DATA_BLOCK "G177M"
TITLE =DBG177M  COOLING / HEATING GERM 4
//COPYRIGHT:    (C) 2009  BUHLER AG, CH-9240 UZWIL, SWITZERLAND
//
//PRODUCT:      WinCoS_BIW01_09
//
//TITLE:        COOLING / HEATING GERM 4
//                Machine group DB
//                Maschinengruppen-DB
//
//-------------------------------------------------------------------------
//
//IDENT:        AUTHOR:             DEPT:             DATE:
//
//P01_DB277.1.0 K.Renz              CSB41             13.Jan.2010
//              1st Release
//
//-------------------------------------------------------------------------
//
//PURPOSE:
//
//MANUAL :
//
//RESTRICTIONS:
//
//-------------------------------------------------------------------------
AUTHOR : KR
FAMILY : USW
NAME : DBG177M
VERSION : 0.0

"G177M_Code"
BEGIN
   Gr.FcCode := 0;
   Gr.Spare2 := 0;
   Gr.Spare4 := 0;
   Gr.Spare6 := 0;
   Gr.OutEmptyingTime := 0;
   Gr.ChangeBit.spare := B#16#0;
   Gr.ChangeBit.CBit1 := FALSE;
   Gr.ChangeBit.CBit2 := FALSE;
   Gr.ChangeBit.CBit3 := FALSE;
   Gr.ChangeBit.CBit4 := FALSE;
   Gr.StCode := 0;
   Gr.InEnableGr := FALSE;
   Gr.CmdContinue := FALSE;
   Gr.CmdRestartIdling := FALSE;
   Gr.InReleaseEmptyingTime := FALSE;
   Gr.InFeeding := FALSE;
   Gr.InOutAutostartMan := FALSE;
   Gr.InPreStart := FALSE;
   Gr.CmdManualOff := FALSE;
   Gr.CmdOff := FALSE;
   Gr.CmdOn := FALSE;
   Gr.CmdNext := FALSE;
   Gr.CmdFaultReset := FALSE;
   Gr.InOccupied := FALSE;
   Gr.InManual := FALSE;
   Gr.InLoadedSec := FALSE;
   Gr.InSeqStop := FALSE;
   Gr.ModePassive := FALSE;
   Gr.ModeActive := FALSE;
   Gr.ModeIdling := FALSE;
   Gr.spare163 := FALSE;
   Gr.spare164 := FALSE;
   Gr.spare165 := FALSE;
   Gr.spare166 := FALSE;
   Gr.spare167 := FALSE;
   Gr.StStopped := FALSE;
   Gr.StStarting := FALSE;
   Gr.StStarted := FALSE;
   Gr.StStopping := FALSE;
   Gr.StFault := FALSE;
   Gr.OutLoaded := FALSE;
   Gr.OutWarning := FALSE;
   Gr.OutFeeding := FALSE;
   Gr.OutEnableEl := FALSE;
   Gr.OutEnable1 := FALSE;
   Gr.OutHWStop := FALSE;
   Gr.OutDPFault := FALSE;
   Gr.OutAutostart := FALSE;
   Gr.OutManual := FALSE;
   Gr.OutHornOn := FALSE;
   Gr.OutEnablePrevGr := FALSE;
   Gr.VarStopped := FALSE;
   Gr.VarStarted := FALSE;
   Gr.VarFault := FALSE;
   Gr.VarStartwarning := FALSE;
   Gr.VarFlag1s := FALSE;
   Gr.OutEmptyingTimeDone := FALSE;
   Gr.OutNewWay := FALSE;
   Gr.OutSeqStop := FALSE;
   Gr.OutIdlingTime := 0;
   Gr.InCodePreselect := 0;
   Gr.InLine := 3;
   Gr.InCode := 0;
   Gr.OutCode := 0;
   Gr.Par.ParObjectNo := 17700;
   Gr.Par.ParMgr := TRUE;
   Gr.Par.ParWgr := FALSE;
   Gr.Par.ParGgr := FALSE;
   Gr.Par.ParHornCode := 5;
   Gr.Par.ParIdling := 2;
   Gr.Par.ParEmptyingTime := 0;
   Gr.Par.Para1_0 := FALSE;
   Gr.Par.Para1_1 := FALSE;
   Gr.Par.Para1_2 := FALSE;
   Gr.Par.Para1_3 := FALSE;
   Gr.Par.Para1_4 := FALSE;
   Gr.Par.Para1_5 := FALSE;
   Gr.Par.Para1_6 := FALSE;
   Gr.Par.Para1_7 := FALSE;
   Gr.Par.Para1_8 := FALSE;
   Gr.Par.Para1_9 := FALSE;
   Gr.Par.Para1_10 := FALSE;
   Gr.Par.Para1_11 := FALSE;
   Gr.Par.Para1_12 := FALSE;
   Gr.Par.Para1_13 := FALSE;
   Gr.Par.Para1_14 := FALSE;
   Gr.Par.Para1_15 := FALSE;
   Gr.Par.Para2 := 0;
   Gr.Par.Para3 := 0;
   Gr.Par.Para4 := 0;
   Gr.Par.Para5 := 0;
   InOutValue1 := L#0;
   InOutValue2 := L#0;
   OutWayConflict := FALSE;
   OutSelectionOk := FALSE;
   CmdNewValue := FALSE;
   CmdNewJob := FALSE;
   OutCodeOK := FALSE;
   InEndOfJob := FALSE;
   staWayOk := FALSE;
   EdgeStartRelease := FALSE;
   USW8 := FALSE;
   USW9 := FALSE;
   USW10 := FALSE;
   USW11 := FALSE;
   USW12 := FALSE;
   USW13 := FALSE;
   USW14 := FALSE;
   USW15 := FALSE;
   A_2445_QXV21.StCode := 0;
   A_2445_QXV21.InEnableRev := FALSE;
   A_2445_QXV21.InEnableFwd := FALSE;
   A_2445_QXV21.InSlow := FALSE;
   A_2445_QXV21.InpRunSlow := FALSE;
   A_2445_QXV21.InpRunFast := FALSE;
   A_2445_QXV21.InpRunRev := FALSE;
   A_2445_QXV21.InpRunFwd := FALSE;
   A_2445_QXV21.InpFaultDev := FALSE;
   A_2445_QXV21.CmdOff := FALSE;
   A_2445_QXV21.CmdOn := FALSE;
   A_2445_QXV21.CmdNext := FALSE;
   A_2445_QXV21.CmdFaultReset := FALSE;
   A_2445_QXV21.InLocal := FALSE;
   A_2445_QXV21.InManual := FALSE;
   A_2445_QXV21.InReport := FALSE;
   A_2445_QXV21.InSeqStop := FALSE;
   A_2445_QXV21.InHWStop := FALSE;
   A_2445_QXV21.InDPFault := FALSE;
   A_2445_QXV21.OutIdling := FALSE;
   A_2445_QXV21.OutpRunSlow := FALSE;
   A_2445_QXV21.OutpRunFast := FALSE;
   A_2445_QXV21.OutpRunRev := FALSE;
   A_2445_QXV21.OutpRunFwd := FALSE;
   A_2445_QXV21.OutpFaultReset := FALSE;
   A_2445_QXV21.StStopped := FALSE;
   A_2445_QXV21.StStarting := FALSE;
   A_2445_QXV21.StStartedFwd := FALSE;
   A_2445_QXV21.StStopping := FALSE;
   A_2445_QXV21.StFault := FALSE;
   A_2445_QXV21.StStartedRev := FALSE;
   A_2445_QXV21.InOutManSlow := FALSE;
   A_2445_QXV21.InOutManRev := FALSE;
   A_2445_QXV21.OutAlarmNrLog := 0;
   A_2445_QXV21.Par.ParObjectNo := 17701;
   A_2445_QXV21.Par.ParMsgType := 7053;
   A_2445_QXV21.Par.ParHornCode := 5;
   A_2445_QXV21.Par.ParLogOff := FALSE;
   A_2445_QXV21.Par.ParManual := TRUE;
   A_2445_QXV21.Par.ParRestartDelay := FALSE;
   A_2445_QXV21.Par.Par2Speed := FALSE;
   A_2445_QXV21.Par.ParHeavyStartup := FALSE;
   A_2445_QXV21.Par.spare45 := FALSE;
   A_2445_QXV21.Par.spare46 := FALSE;
   A_2445_QXV21.Par.OutEdgeFaultReset := FALSE;
   A_2445_QXV21.Par.OutDelayFault := FALSE;
   A_2445_QXV21.Par.OutFlagFaultDev := FALSE;
   A_2445_QXV21.Par.ParMonTime := 20;
   A_2445_QXV21.Par.ParStartingTime := 20;
   A_2445_QXV21.Par.ParStoppingTime := 0;
   A_2445_QXV21.Par.ParIdlingTime := 0;
   A_2445_QXV21.Par.ParDelayTime := 10;
   A_2445_QXV21.Par.OutMonTime := 0;
   A_2445_QXV21.Par.OutTransitionTime := 0;
   A_2445_QXV21.Par.OutDelayTime := 0;
   A_2445_QXV21.Par.InOutManPulseLen := 0;
   A_2445_QXV21AI.StCode := 2;
   A_2445_QXV21AI.InMonLL := FALSE;
   A_2445_QXV21AI.InMonL := FALSE;
   A_2445_QXV21AI.InMonMid := FALSE;
   A_2445_QXV21AI.InMonH := FALSE;
   A_2445_QXV21AI.InMonHH := FALSE;
   A_2445_QXV21AI.spare0205 := FALSE;
   A_2445_QXV21AI.InpFaultAI := FALSE;
   A_2445_QXV21AI.InpFaultDev := FALSE;
   A_2445_QXV21AI.InHWStop := FALSE;
   A_2445_QXV21AI.InDPFault := FALSE;
   A_2445_QXV21AI.InDisable := FALSE;
   A_2445_QXV21AI.CmdFaultReset := FALSE;
   A_2445_QXV21AI.InLocal := FALSE;
   A_2445_QXV21AI.spare0305 := FALSE;
   A_2445_QXV21AI.InReport := FALSE;
   A_2445_QXV21AI.spare0307 := FALSE;
   A_2445_QXV21AI.OutLL := FALSE;
   A_2445_QXV21AI.OutL := FALSE;
   A_2445_QXV21AI.OutH := FALSE;
   A_2445_QXV21AI.OutHH := FALSE;
   A_2445_QXV21AI.OutOverflow := FALSE;
   A_2445_QXV21AI.spare0405 := FALSE;
   A_2445_QXV21AI.OutFaultAI := FALSE;
   A_2445_QXV21AI.spare0407 := FALSE;
   A_2445_QXV21AI.StLL := FALSE;
   A_2445_QXV21AI.StL := FALSE;
   A_2445_QXV21AI.StMid := FALSE;
   A_2445_QXV21AI.StH := FALSE;
   A_2445_QXV21AI.StHH := FALSE;
   A_2445_QXV21AI.StFaultAI := FALSE;
   A_2445_QXV21AI.OutWarning := FALSE;
   A_2445_QXV21AI.OutFaulted := FALSE;
   A_2445_QXV21AI.InpValue := 0;
   A_2445_QXV21AI.OutValuePc := 0;
   A_2445_QXV21AI.OutValueUnits := L#0;
   A_2445_QXV21AI.Msg.WarningDoneLL := FALSE;
   A_2445_QXV21AI.Msg.WarningDoneL := FALSE;
   A_2445_QXV21AI.Msg.WarningDoneMid := FALSE;
   A_2445_QXV21AI.Msg.WarningDoneH := FALSE;
   A_2445_QXV21AI.Msg.WarningDoneHH := FALSE;
   A_2445_QXV21AI.Msg.FaultDoneLL := FALSE;
   A_2445_QXV21AI.Msg.FaultDoneL := FALSE;
   A_2445_QXV21AI.Msg.FaultDoneMid := FALSE;
   A_2445_QXV21AI.Msg.FaultDoneH := FALSE;
   A_2445_QXV21AI.Msg.FaultDoneHH := FALSE;
   A_2445_QXV21AI.Msg.FaultDoneDev := FALSE;
   A_2445_QXV21AI.Msg.FaultDoneAI := FALSE;
   A_2445_QXV21AI.OutAlarmNrLog := 0;
   A_2445_QXV21AI.Par.ParObjectNo := 17702;
   A_2445_QXV21AI.Par.ParMsgType := 7252;
   A_2445_QXV21AI.Par.ParHornCode := 0;
   A_2445_QXV21AI.Par.ParLogOff := FALSE;
   A_2445_QXV21AI.Par.ParSpare0401 := FALSE;
   A_2445_QXV21AI.Par.ParValueByUser := FALSE;
   A_2445_QXV21AI.Par.ParLimitsPc := TRUE;
   A_2445_QXV21AI.Par.ParWago := FALSE;
   A_2445_QXV21AI.Par.ParNoHornByWarning := FALSE;
   A_2445_QXV21AI.Par.ParWarningLL := FALSE;
   A_2445_QXV21AI.Par.ParWarningL := FALSE;
   A_2445_QXV21AI.Par.ParWarningMid := FALSE;
   A_2445_QXV21AI.Par.ParWarningH := FALSE;
   A_2445_QXV21AI.Par.ParWarningHH := FALSE;
   A_2445_QXV21AI.Par.ParPreAlarmLL := FALSE;
   A_2445_QXV21AI.Par.ParPreAlarmL := FALSE;
   A_2445_QXV21AI.Par.ParPreAlarmMid := FALSE;
   A_2445_QXV21AI.Par.ParPreAlarmH := FALSE;
   A_2445_QXV21AI.Par.ParPreAlarmHH := FALSE;
   A_2445_QXV21AI.Par.ParUnitsByZeroDigit := L#0;
   A_2445_QXV21AI.Par.ParUnitsByMaxDigit := L#10000;
   A_2445_QXV21AI.Par.ParUnitsBy100Pc := L#10000;
   A_2445_QXV21AI.Par.ParLimitLL := L#0;
   A_2445_QXV21AI.Par.ParLimitL := L#2000;
   A_2445_QXV21AI.Par.ParLimitH := L#8000;
   A_2445_QXV21AI.Par.ParLimitHH := L#10000;
   A_2445_QXV21AI.Par.ParMonTimeLL := 0;
   A_2445_QXV21AI.Par.ParMonTimeL := 50;
   A_2445_QXV21AI.Par.ParMonTimeMid := 0;
   A_2445_QXV21AI.Par.ParMonTimeH := 30;
   A_2445_QXV21AI.Par.ParMonTimeHH := 0;
   A_2445_QXV21AI.Par.ParDelayTimeDown := 10;
   A_2445_QXV21AI.Par.ParDelayTimeUp := 10;
   A_2445_QXV21AI.Par.ParDelayTime := 0;
   A_2445_QXV21AI.Par.OutMonTimeLL := 0;
   A_2445_QXV21AI.Par.OutMonTimeL := 50;
   A_2445_QXV21AI.Par.OutMonTimeMid := 0;
   A_2445_QXV21AI.Par.OutMonTimeH := 0;
   A_2445_QXV21AI.Par.OutMonTimeHH := 0;
   A_2445_QXV21AI.Par.OutDelayTimeDown := 0;
   A_2445_QXV21AI.Par.OutDelayTimeUp := 0;
   A_2445_QXV21AI.Par.OutDelayTime := 0;
   A_2445_QXV21AI.Par.Spare66 := 0;
   A_2445_QXV21AO.StCode := 0;
   A_2445_QXV21AO.InDisable := FALSE;
   A_2445_QXV21AO.spare0201 := FALSE;
   A_2445_QXV21AO.spare0202 := FALSE;
   A_2445_QXV21AO.spare0203 := FALSE;
   A_2445_QXV21AO.spare0204 := FALSE;
   A_2445_QXV21AO.spare0205 := FALSE;
   A_2445_QXV21AO.spare0206 := FALSE;
   A_2445_QXV21AO.InpFaultDev := FALSE;
   A_2445_QXV21AO.spare0300 := FALSE;
   A_2445_QXV21AO.spare0301 := FALSE;
   A_2445_QXV21AO.spare0302 := FALSE;
   A_2445_QXV21AO.CmdFaultReset := FALSE;
   A_2445_QXV21AO.InLocal := FALSE;
   A_2445_QXV21AO.InManual := FALSE;
   A_2445_QXV21AO.InReport := FALSE;
   A_2445_QXV21AO.spare0307 := FALSE;
   A_2445_QXV21AO.InHWStop := FALSE;
   A_2445_QXV21AO.InDPFault := FALSE;
   A_2445_QXV21AO.spare0402 := FALSE;
   A_2445_QXV21AO.spare0403 := FALSE;
   A_2445_QXV21AO.spare0404 := FALSE;
   A_2445_QXV21AO.OutpFaultReset := FALSE;
   A_2445_QXV21AO.OutMin := FALSE;
   A_2445_QXV21AO.OutMax := FALSE;
   A_2445_QXV21AO.StOff := FALSE;
   A_2445_QXV21AO.spare0501 := FALSE;
   A_2445_QXV21AO.StOn := FALSE;
   A_2445_QXV21AO.spare0503 := FALSE;
   A_2445_QXV21AO.StFault := FALSE;
   A_2445_QXV21AO.OutpValue := 0;
   A_2445_QXV21AO.InOutValuePc := 0;
   A_2445_QXV21AO.InOutValueUnits := L#0;
   A_2445_QXV21AO.ASW := L#0;
   A_2445_QXV21AO.OutAlarmNrLog := 0;
   A_2445_QXV21AO.Par.ParObjectNo := 17703;
   A_2445_QXV21AO.Par.ParMsgType := 7241;
   A_2445_QXV21AO.Par.ParHornCode := 5;
   A_2445_QXV21AO.Par.ParLogOff := FALSE;
   A_2445_QXV21AO.Par.ParFU := FALSE;
   A_2445_QXV21AO.Par.ParValuePc := TRUE;
   A_2445_QXV21AO.Par.ParLimitsPc := TRUE;
   A_2445_QXV21AO.Par.ParWago := FALSE;
   A_2445_QXV21AO.Par.ParUnitsByZeroDigit := L#0;
   A_2445_QXV21AO.Par.ParUnitsByMaxDigit := L#27648;
   A_2445_QXV21AO.Par.ParUnitsBy100Pc := L#10000;
   A_2445_QXV21AO.Par.ParLimitMin := L#0;
   A_2445_QXV21AO.Par.ParLimitMax := L#27648;
   A_2445_QXV21AO.Par.ParDelayTime := 30;
   A_2445_QXV21AO.Par.OutDelayTime := 0;
   A_2445_QXV21I1.StCode := 0;
   A_2445_QXV21I1.InMonTrue := FALSE;
   A_2445_QXV21I1.InMonFalse := FALSE;
   A_2445_QXV21I1.InPreAlarmTrue := FALSE;
   A_2445_QXV21I1.InPreAlarmFalse := FALSE;
   A_2445_QXV21I1.InStopTrueTime := FALSE;
   A_2445_QXV21I1.InStopFalseTime := FALSE;
   A_2445_QXV21I1.InpTrue := FALSE;
   A_2445_QXV21I1.InpFaultDev := FALSE;
   A_2445_QXV21I1.CmdRstTrueTime := FALSE;
   A_2445_QXV21I1.CmdRstFalseTime := FALSE;
   A_2445_QXV21I1.CmdRunTimeoutTime := FALSE;
   A_2445_QXV21I1.CmdFaultReset := FALSE;
   A_2445_QXV21I1.InLocal := FALSE;
   A_2445_QXV21I1.spare0305 := FALSE;
   A_2445_QXV21I1.InReport := FALSE;
   A_2445_QXV21I1.OutTimeoutTime := FALSE;
   A_2445_QXV21I1.InHWStop := FALSE;
   A_2445_QXV21I1.InDPFault := FALSE;
   A_2445_QXV21I1.OutPreAlarmTrue := FALSE;
   A_2445_QXV21I1.OutPreAlarmFalse := FALSE;
   A_2445_QXV21I1.OutFlagPos := FALSE;
   A_2445_QXV21I1.OutFlagNeg := FALSE;
   A_2445_QXV21I1.OutpFaultReset := FALSE;
   A_2445_QXV21I1.OutTrue := FALSE;
   A_2445_QXV21I1.StFalse := FALSE;
   A_2445_QXV21I1.StCtoTrue := FALSE;
   A_2445_QXV21I1.StTrue := FALSE;
   A_2445_QXV21I1.StCtoFalse := FALSE;
   A_2445_QXV21I1.StFault := FALSE;
   A_2445_QXV21I1.OutAlarmNrLog := 0;
   A_2445_QXV21I1.Par.ParObjectNo := 17704;
   A_2445_QXV21I1.Par.ParMsgType := 7163;
   A_2445_QXV21I1.Par.ParHornCode := 5;
   A_2445_QXV21I1.Par.ParLogOff := FALSE;
   A_2445_QXV21I1.Par.spare0401 := FALSE;
   A_2445_QXV21I1.Par.Par2WorkingCond := FALSE;
   A_2445_QXV21I1.Par.ParFaultRetry := FALSE;
   A_2445_QXV21I1.Par.ParBinLevel := FALSE;
   A_2445_QXV21I1.Par.ParDelayChange := 20;
   A_2445_QXV21I1.Par.ParDelayTrue := 10;
   A_2445_QXV21I1.Par.ParDelayFalse := 0;
   A_2445_QXV21I1.Par.ParTimeoutTrue := 0;
   A_2445_QXV21I1.Par.ParTimeoutFalse := 0;
   A_2445_QXV21I1.Par.OutMonTime := 0;
   A_2445_QXV21I1.Par.OutTransitionTime := 0;
   A_2445_QXV21I1.Par.OutMonTrue := FALSE;
   A_2445_QXV21I1.Par.OutMonFalse := FALSE;
   A_2445_QXV21I1.Par.OutFlagFaultDev := FALSE;
   A_2445_QXV21I1.Par.OutDelayTime := 20;
   A_2445_QXV21I2.StCode := 0;
   A_2445_QXV21I2.InMonTrue := FALSE;
   A_2445_QXV21I2.InMonFalse := FALSE;
   A_2445_QXV21I2.InPreAlarmTrue := FALSE;
   A_2445_QXV21I2.InPreAlarmFalse := FALSE;
   A_2445_QXV21I2.InStopTrueTime := FALSE;
   A_2445_QXV21I2.InStopFalseTime := FALSE;
   A_2445_QXV21I2.InpTrue := FALSE;
   A_2445_QXV21I2.InpFaultDev := FALSE;
   A_2445_QXV21I2.CmdRstTrueTime := FALSE;
   A_2445_QXV21I2.CmdRstFalseTime := FALSE;
   A_2445_QXV21I2.CmdRunTimeoutTime := FALSE;
   A_2445_QXV21I2.CmdFaultReset := FALSE;
   A_2445_QXV21I2.InLocal := FALSE;
   A_2445_QXV21I2.spare0305 := FALSE;
   A_2445_QXV21I2.InReport := FALSE;
   A_2445_QXV21I2.OutTimeoutTime := FALSE;
   A_2445_QXV21I2.InHWStop := FALSE;
   A_2445_QXV21I2.InDPFault := FALSE;
   A_2445_QXV21I2.OutPreAlarmTrue := FALSE;
   A_2445_QXV21I2.OutPreAlarmFalse := FALSE;
   A_2445_QXV21I2.OutFlagPos := FALSE;
   A_2445_QXV21I2.OutFlagNeg := FALSE;
   A_2445_QXV21I2.OutpFaultReset := FALSE;
   A_2445_QXV21I2.OutTrue := FALSE;
   A_2445_QXV21I2.StFalse := FALSE;
   A_2445_QXV21I2.StCtoTrue := FALSE;
   A_2445_QXV21I2.StTrue := FALSE;
   A_2445_QXV21I2.StCtoFalse := FALSE;
   A_2445_QXV21I2.StFault := FALSE;
   A_2445_QXV21I2.OutAlarmNrLog := 0;
   A_2445_QXV21I2.Par.ParObjectNo := 17705;
   A_2445_QXV21I2.Par.ParMsgType := 7163;
   A_2445_QXV21I2.Par.ParHornCode := 5;
   A_2445_QXV21I2.Par.ParLogOff := FALSE;
   A_2445_QXV21I2.Par.spare0401 := FALSE;
   A_2445_QXV21I2.Par.Par2WorkingCond := FALSE;
   A_2445_QXV21I2.Par.ParFaultRetry := FALSE;
   A_2445_QXV21I2.Par.ParBinLevel := FALSE;
   A_2445_QXV21I2.Par.ParDelayChange := 20;
   A_2445_QXV21I2.Par.ParDelayTrue := 10;
   A_2445_QXV21I2.Par.ParDelayFalse := 0;
   A_2445_QXV21I2.Par.ParTimeoutTrue := 0;
   A_2445_QXV21I2.Par.ParTimeoutFalse := 0;
   A_2445_QXV21I2.Par.OutMonTime := 0;
   A_2445_QXV21I2.Par.OutTransitionTime := 0;
   A_2445_QXV21I2.Par.OutMonTrue := FALSE;
   A_2445_QXV21I2.Par.OutMonFalse := FALSE;
   A_2445_QXV21I2.Par.OutFlagFaultDev := FALSE;
   A_2445_QXV21I2.Par.OutDelayTime := 20;
   A_2445_QXV31.StCode := 0;
   A_2445_QXV31.InEnableRev := FALSE;
   A_2445_QXV31.InEnableFwd := FALSE;
   A_2445_QXV31.InSlow := FALSE;
   A_2445_QXV31.InpRunSlow := FALSE;
   A_2445_QXV31.InpRunFast := FALSE;
   A_2445_QXV31.InpRunRev := FALSE;
   A_2445_QXV31.InpRunFwd := FALSE;
   A_2445_QXV31.InpFaultDev := FALSE;
   A_2445_QXV31.CmdOff := FALSE;
   A_2445_QXV31.CmdOn := FALSE;
   A_2445_QXV31.CmdNext := FALSE;
   A_2445_QXV31.CmdFaultReset := FALSE;
   A_2445_QXV31.InLocal := FALSE;
   A_2445_QXV31.InManual := FALSE;
   A_2445_QXV31.InReport := FALSE;
   A_2445_QXV31.InSeqStop := FALSE;
   A_2445_QXV31.InHWStop := FALSE;
   A_2445_QXV31.InDPFault := FALSE;
   A_2445_QXV31.OutIdling := FALSE;
   A_2445_QXV31.OutpRunSlow := FALSE;
   A_2445_QXV31.OutpRunFast := FALSE;
   A_2445_QXV31.OutpRunRev := FALSE;
   A_2445_QXV31.OutpRunFwd := FALSE;
   A_2445_QXV31.OutpFaultReset := FALSE;
   A_2445_QXV31.StStopped := FALSE;
   A_2445_QXV31.StStarting := FALSE;
   A_2445_QXV31.StStartedFwd := FALSE;
   A_2445_QXV31.StStopping := FALSE;
   A_2445_QXV31.StFault := FALSE;
   A_2445_QXV31.StStartedRev := FALSE;
   A_2445_QXV31.InOutManSlow := FALSE;
   A_2445_QXV31.InOutManRev := FALSE;
   A_2445_QXV31.OutAlarmNrLog := 0;
   A_2445_QXV31.Par.ParObjectNo := 17706;
   A_2445_QXV31.Par.ParMsgType := 7053;
   A_2445_QXV31.Par.ParHornCode := 5;
   A_2445_QXV31.Par.ParLogOff := FALSE;
   A_2445_QXV31.Par.ParManual := TRUE;
   A_2445_QXV31.Par.ParRestartDelay := FALSE;
   A_2445_QXV31.Par.Par2Speed := FALSE;
   A_2445_QXV31.Par.ParHeavyStartup := FALSE;
   A_2445_QXV31.Par.spare45 := FALSE;
   A_2445_QXV31.Par.spare46 := FALSE;
   A_2445_QXV31.Par.OutEdgeFaultReset := FALSE;
   A_2445_QXV31.Par.OutDelayFault := FALSE;
   A_2445_QXV31.Par.OutFlagFaultDev := FALSE;
   A_2445_QXV31.Par.ParMonTime := 20;
   A_2445_QXV31.Par.ParStartingTime := 20;
   A_2445_QXV31.Par.ParStoppingTime := 0;
   A_2445_QXV31.Par.ParIdlingTime := 0;
   A_2445_QXV31.Par.ParDelayTime := 10;
   A_2445_QXV31.Par.OutMonTime := 0;
   A_2445_QXV31.Par.OutTransitionTime := 0;
   A_2445_QXV31.Par.OutDelayTime := 0;
   A_2445_QXV31.Par.InOutManPulseLen := 0;
   A_2445_QXV31AI.StCode := 0;
   A_2445_QXV31AI.InMonLL := FALSE;
   A_2445_QXV31AI.InMonL := FALSE;
   A_2445_QXV31AI.InMonMid := FALSE;
   A_2445_QXV31AI.InMonH := FALSE;
   A_2445_QXV31AI.InMonHH := FALSE;
   A_2445_QXV31AI.spare0205 := FALSE;
   A_2445_QXV31AI.InpFaultAI := FALSE;
   A_2445_QXV31AI.InpFaultDev := FALSE;
   A_2445_QXV31AI.InHWStop := FALSE;
   A_2445_QXV31AI.InDPFault := FALSE;
   A_2445_QXV31AI.InDisable := FALSE;
   A_2445_QXV31AI.CmdFaultReset := FALSE;
   A_2445_QXV31AI.InLocal := FALSE;
   A_2445_QXV31AI.spare0305 := FALSE;
   A_2445_QXV31AI.InReport := FALSE;
   A_2445_QXV31AI.spare0307 := FALSE;
   A_2445_QXV31AI.OutLL := FALSE;
   A_2445_QXV31AI.OutL := FALSE;
   A_2445_QXV31AI.OutH := FALSE;
   A_2445_QXV31AI.OutHH := FALSE;
   A_2445_QXV31AI.OutOverflow := FALSE;
   A_2445_QXV31AI.spare0405 := FALSE;
   A_2445_QXV31AI.OutFaultAI := FALSE;
   A_2445_QXV31AI.spare0407 := FALSE;
   A_2445_QXV31AI.StLL := FALSE;
   A_2445_QXV31AI.StL := FALSE;
   A_2445_QXV31AI.StMid := FALSE;
   A_2445_QXV31AI.StH := FALSE;
   A_2445_QXV31AI.StHH := FALSE;
   A_2445_QXV31AI.StFaultAI := FALSE;
   A_2445_QXV31AI.OutWarning := FALSE;
   A_2445_QXV31AI.OutFaulted := FALSE;
   A_2445_QXV31AI.InpValue := 0;
   A_2445_QXV31AI.OutValuePc := 0;
   A_2445_QXV31AI.OutValueUnits := L#0;
   A_2445_QXV31AI.Msg.WarningDoneLL := FALSE;
   A_2445_QXV31AI.Msg.WarningDoneL := FALSE;
   A_2445_QXV31AI.Msg.WarningDoneMid := FALSE;
   A_2445_QXV31AI.Msg.WarningDoneH := FALSE;
   A_2445_QXV31AI.Msg.WarningDoneHH := FALSE;
   A_2445_QXV31AI.Msg.FaultDoneLL := FALSE;
   A_2445_QXV31AI.Msg.FaultDoneL := FALSE;
   A_2445_QXV31AI.Msg.FaultDoneMid := FALSE;
   A_2445_QXV31AI.Msg.FaultDoneH := FALSE;
   A_2445_QXV31AI.Msg.FaultDoneHH := FALSE;
   A_2445_QXV31AI.Msg.FaultDoneDev := FALSE;
   A_2445_QXV31AI.Msg.FaultDoneAI := FALSE;
   A_2445_QXV31AI.OutAlarmNrLog := 0;
   A_2445_QXV31AI.Par.ParObjectNo := 17707;
   A_2445_QXV31AI.Par.ParMsgType := 7252;
   A_2445_QXV31AI.Par.ParHornCode := 5;
   A_2445_QXV31AI.Par.ParLogOff := FALSE;
   A_2445_QXV31AI.Par.ParSpare0401 := FALSE;
   A_2445_QXV31AI.Par.ParValueByUser := FALSE;
   A_2445_QXV31AI.Par.ParLimitsPc := TRUE;
   A_2445_QXV31AI.Par.ParWago := FALSE;
   A_2445_QXV31AI.Par.ParNoHornByWarning := FALSE;
   A_2445_QXV31AI.Par.ParWarningLL := FALSE;
   A_2445_QXV31AI.Par.ParWarningL := FALSE;
   A_2445_QXV31AI.Par.ParWarningMid := FALSE;
   A_2445_QXV31AI.Par.ParWarningH := FALSE;
   A_2445_QXV31AI.Par.ParWarningHH := FALSE;
   A_2445_QXV31AI.Par.ParPreAlarmLL := FALSE;
   A_2445_QXV31AI.Par.ParPreAlarmL := FALSE;
   A_2445_QXV31AI.Par.ParPreAlarmMid := FALSE;
   A_2445_QXV31AI.Par.ParPreAlarmH := FALSE;
   A_2445_QXV31AI.Par.ParPreAlarmHH := FALSE;
   A_2445_QXV31AI.Par.ParUnitsByZeroDigit := L#0;
   A_2445_QXV31AI.Par.ParUnitsByMaxDigit := L#10000;
   A_2445_QXV31AI.Par.ParUnitsBy100Pc := L#10000;
   A_2445_QXV31AI.Par.ParLimitLL := L#0;
   A_2445_QXV31AI.Par.ParLimitL := L#2000;
   A_2445_QXV31AI.Par.ParLimitH := L#8000;
   A_2445_QXV31AI.Par.ParLimitHH := L#10000;
   A_2445_QXV31AI.Par.ParMonTimeLL := 0;
   A_2445_QXV31AI.Par.ParMonTimeL := 50;
   A_2445_QXV31AI.Par.ParMonTimeMid := 0;
   A_2445_QXV31AI.Par.ParMonTimeH := 30;
   A_2445_QXV31AI.Par.ParMonTimeHH := 0;
   A_2445_QXV31AI.Par.ParDelayTimeDown := 10;
   A_2445_QXV31AI.Par.ParDelayTimeUp := 10;
   A_2445_QXV31AI.Par.ParDelayTime := 0;
   A_2445_QXV31AI.Par.OutMonTimeLL := 0;
   A_2445_QXV31AI.Par.OutMonTimeL := 50;
   A_2445_QXV31AI.Par.OutMonTimeMid := 0;
   A_2445_QXV31AI.Par.OutMonTimeH := 0;
   A_2445_QXV31AI.Par.OutMonTimeHH := 0;
   A_2445_QXV31AI.Par.OutDelayTimeDown := 0;
   A_2445_QXV31AI.Par.OutDelayTimeUp := 0;
   A_2445_QXV31AI.Par.OutDelayTime := 0;
   A_2445_QXV31AI.Par.Spare66 := 0;
   A_2445_QXV31AO.StCode := 0;
   A_2445_QXV31AO.InDisable := FALSE;
   A_2445_QXV31AO.spare0201 := FALSE;
   A_2445_QXV31AO.spare0202 := FALSE;
   A_2445_QXV31AO.spare0203 := FALSE;
   A_2445_QXV31AO.spare0204 := FALSE;
   A_2445_QXV31AO.spare0205 := FALSE;
   A_2445_QXV31AO.spare0206 := FALSE;
   A_2445_QXV31AO.InpFaultDev := FALSE;
   A_2445_QXV31AO.spare0300 := FALSE;
   A_2445_QXV31AO.spare0301 := FALSE;
   A_2445_QXV31AO.spare0302 := FALSE;
   A_2445_QXV31AO.CmdFaultReset := FALSE;
   A_2445_QXV31AO.InLocal := FALSE;
   A_2445_QXV31AO.InManual := FALSE;
   A_2445_QXV31AO.InReport := FALSE;
   A_2445_QXV31AO.spare0307 := FALSE;
   A_2445_QXV31AO.InHWStop := FALSE;
   A_2445_QXV31AO.InDPFault := FALSE;
   A_2445_QXV31AO.spare0402 := FALSE;
   A_2445_QXV31AO.spare0403 := FALSE;
   A_2445_QXV31AO.spare0404 := FALSE;
   A_2445_QXV31AO.OutpFaultReset := FALSE;
   A_2445_QXV31AO.OutMin := FALSE;
   A_2445_QXV31AO.OutMax := TRUE;
   A_2445_QXV31AO.StOff := FALSE;
   A_2445_QXV31AO.spare0501 := FALSE;
   A_2445_QXV31AO.StOn := TRUE;
   A_2445_QXV31AO.spare0503 := FALSE;
   A_2445_QXV31AO.StFault := FALSE;
   A_2445_QXV31AO.OutpValue := 0;
   A_2445_QXV31AO.InOutValuePc := 0;
   A_2445_QXV31AO.InOutValueUnits := L#0;
   A_2445_QXV31AO.ASW := L#0;
   A_2445_QXV31AO.OutAlarmNrLog := 0;
   A_2445_QXV31AO.Par.ParObjectNo := 17708;
   A_2445_QXV31AO.Par.ParMsgType := 7241;
   A_2445_QXV31AO.Par.ParHornCode := 5;
   A_2445_QXV31AO.Par.ParLogOff := FALSE;
   A_2445_QXV31AO.Par.ParFU := FALSE;
   A_2445_QXV31AO.Par.ParValuePc := TRUE;
   A_2445_QXV31AO.Par.ParLimitsPc := TRUE;
   A_2445_QXV31AO.Par.ParWago := FALSE;
   A_2445_QXV31AO.Par.ParUnitsByZeroDigit := L#0;
   A_2445_QXV31AO.Par.ParUnitsByMaxDigit := L#27648;
   A_2445_QXV31AO.Par.ParUnitsBy100Pc := L#10000;
   A_2445_QXV31AO.Par.ParLimitMin := L#0;
   A_2445_QXV31AO.Par.ParLimitMax := L#27648;
   A_2445_QXV31AO.Par.ParDelayTime := 30;
   A_2445_QXV31AO.Par.OutDelayTime := 0;
   A_2445_QXV31I1.StCode := 0;
   A_2445_QXV31I1.InMonTrue := FALSE;
   A_2445_QXV31I1.InMonFalse := FALSE;
   A_2445_QXV31I1.InPreAlarmTrue := FALSE;
   A_2445_QXV31I1.InPreAlarmFalse := FALSE;
   A_2445_QXV31I1.InStopTrueTime := FALSE;
   A_2445_QXV31I1.InStopFalseTime := FALSE;
   A_2445_QXV31I1.InpTrue := FALSE;
   A_2445_QXV31I1.InpFaultDev := FALSE;
   A_2445_QXV31I1.CmdRstTrueTime := FALSE;
   A_2445_QXV31I1.CmdRstFalseTime := FALSE;
   A_2445_QXV31I1.CmdRunTimeoutTime := FALSE;
   A_2445_QXV31I1.CmdFaultReset := FALSE;
   A_2445_QXV31I1.InLocal := FALSE;
   A_2445_QXV31I1.spare0305 := FALSE;
   A_2445_QXV31I1.InReport := FALSE;
   A_2445_QXV31I1.OutTimeoutTime := FALSE;
   A_2445_QXV31I1.InHWStop := FALSE;
   A_2445_QXV31I1.InDPFault := FALSE;
   A_2445_QXV31I1.OutPreAlarmTrue := FALSE;
   A_2445_QXV31I1.OutPreAlarmFalse := FALSE;
   A_2445_QXV31I1.OutFlagPos := FALSE;
   A_2445_QXV31I1.OutFlagNeg := FALSE;
   A_2445_QXV31I1.OutpFaultReset := FALSE;
   A_2445_QXV31I1.OutTrue := FALSE;
   A_2445_QXV31I1.StFalse := FALSE;
   A_2445_QXV31I1.StCtoTrue := FALSE;
   A_2445_QXV31I1.StTrue := FALSE;
   A_2445_QXV31I1.StCtoFalse := FALSE;
   A_2445_QXV31I1.StFault := FALSE;
   A_2445_QXV31I1.OutAlarmNrLog := 0;
   A_2445_QXV31I1.Par.ParObjectNo := 17709;
   A_2445_QXV31I1.Par.ParMsgType := 7163;
   A_2445_QXV31I1.Par.ParHornCode := 5;
   A_2445_QXV31I1.Par.ParLogOff := FALSE;
   A_2445_QXV31I1.Par.spare0401 := FALSE;
   A_2445_QXV31I1.Par.Par2WorkingCond := FALSE;
   A_2445_QXV31I1.Par.ParFaultRetry := FALSE;
   A_2445_QXV31I1.Par.ParBinLevel := FALSE;
   A_2445_QXV31I1.Par.ParDelayChange := 20;
   A_2445_QXV31I1.Par.ParDelayTrue := 10;
   A_2445_QXV31I1.Par.ParDelayFalse := 0;
   A_2445_QXV31I1.Par.ParTimeoutTrue := 0;
   A_2445_QXV31I1.Par.ParTimeoutFalse := 0;
   A_2445_QXV31I1.Par.OutMonTime := 0;
   A_2445_QXV31I1.Par.OutTransitionTime := 0;
   A_2445_QXV31I1.Par.OutMonTrue := FALSE;
   A_2445_QXV31I1.Par.OutMonFalse := FALSE;
   A_2445_QXV31I1.Par.OutFlagFaultDev := FALSE;
   A_2445_QXV31I1.Par.OutDelayTime := 0;
   A_2445_QXV31I2.StCode := 0;
   A_2445_QXV31I2.InMonTrue := FALSE;
   A_2445_QXV31I2.InMonFalse := FALSE;
   A_2445_QXV31I2.InPreAlarmTrue := FALSE;
   A_2445_QXV31I2.InPreAlarmFalse := FALSE;
   A_2445_QXV31I2.InStopTrueTime := FALSE;
   A_2445_QXV31I2.InStopFalseTime := FALSE;
   A_2445_QXV31I2.InpTrue := FALSE;
   A_2445_QXV31I2.InpFaultDev := FALSE;
   A_2445_QXV31I2.CmdRstTrueTime := FALSE;
   A_2445_QXV31I2.CmdRstFalseTime := FALSE;
   A_2445_QXV31I2.CmdRunTimeoutTime := FALSE;
   A_2445_QXV31I2.CmdFaultReset := FALSE;
   A_2445_QXV31I2.InLocal := FALSE;
   A_2445_QXV31I2.spare0305 := FALSE;
   A_2445_QXV31I2.InReport := FALSE;
   A_2445_QXV31I2.OutTimeoutTime := FALSE;
   A_2445_QXV31I2.InHWStop := FALSE;
   A_2445_QXV31I2.InDPFault := FALSE;
   A_2445_QXV31I2.OutPreAlarmTrue := FALSE;
   A_2445_QXV31I2.OutPreAlarmFalse := FALSE;
   A_2445_QXV31I2.OutFlagPos := FALSE;
   A_2445_QXV31I2.OutFlagNeg := FALSE;
   A_2445_QXV31I2.OutpFaultReset := FALSE;
   A_2445_QXV31I2.OutTrue := FALSE;
   A_2445_QXV31I2.StFalse := FALSE;
   A_2445_QXV31I2.StCtoTrue := FALSE;
   A_2445_QXV31I2.StTrue := FALSE;
   A_2445_QXV31I2.StCtoFalse := FALSE;
   A_2445_QXV31I2.StFault := FALSE;
   A_2445_QXV31I2.OutAlarmNrLog := 0;
   A_2445_QXV31I2.Par.ParObjectNo := 17710;
   A_2445_QXV31I2.Par.ParMsgType := 7163;
   A_2445_QXV31I2.Par.ParHornCode := 0;
   A_2445_QXV31I2.Par.ParLogOff := FALSE;
   A_2445_QXV31I2.Par.spare0401 := FALSE;
   A_2445_QXV31I2.Par.Par2WorkingCond := FALSE;
   A_2445_QXV31I2.Par.ParFaultRetry := FALSE;
   A_2445_QXV31I2.Par.ParBinLevel := FALSE;
   A_2445_QXV31I2.Par.ParDelayChange := 20;
   A_2445_QXV31I2.Par.ParDelayTrue := 10;
   A_2445_QXV31I2.Par.ParDelayFalse := 0;
   A_2445_QXV31I2.Par.ParTimeoutTrue := 0;
   A_2445_QXV31I2.Par.ParTimeoutFalse := 0;
   A_2445_QXV31I2.Par.OutMonTime := 0;
   A_2445_QXV31I2.Par.OutTransitionTime := 0;
   A_2445_QXV31I2.Par.OutMonTrue := FALSE;
   A_2445_QXV31I2.Par.OutMonFalse := FALSE;
   A_2445_QXV31I2.Par.OutFlagFaultDev := FALSE;
   A_2445_QXV31I2.Par.OutDelayTime := 20;
   A_2454_MXZ01.StCode := 0;
   A_2454_MXZ01.InEnableRev := FALSE;
   A_2454_MXZ01.InEnableFwd := FALSE;
   A_2454_MXZ01.InSlow := FALSE;
   A_2454_MXZ01.InpRunSlow := FALSE;
   A_2454_MXZ01.InpRunFast := FALSE;
   A_2454_MXZ01.InpRunRev := FALSE;
   A_2454_MXZ01.InpRunFwd := FALSE;
   A_2454_MXZ01.InpFaultDev := FALSE;
   A_2454_MXZ01.CmdOff := FALSE;
   A_2454_MXZ01.CmdOn := FALSE;
   A_2454_MXZ01.CmdNext := FALSE;
   A_2454_MXZ01.CmdFaultReset := FALSE;
   A_2454_MXZ01.InLocal := FALSE;
   A_2454_MXZ01.InManual := FALSE;
   A_2454_MXZ01.InReport := FALSE;
   A_2454_MXZ01.InSeqStop := FALSE;
   A_2454_MXZ01.InHWStop := FALSE;
   A_2454_MXZ01.InDPFault := FALSE;
   A_2454_MXZ01.OutIdling := FALSE;
   A_2454_MXZ01.OutpRunSlow := FALSE;
   A_2454_MXZ01.OutpRunFast := FALSE;
   A_2454_MXZ01.OutpRunRev := FALSE;
   A_2454_MXZ01.OutpRunFwd := FALSE;
   A_2454_MXZ01.OutpFaultReset := FALSE;
   A_2454_MXZ01.StStopped := FALSE;
   A_2454_MXZ01.StStarting := FALSE;
   A_2454_MXZ01.StStartedFwd := FALSE;
   A_2454_MXZ01.StStopping := FALSE;
   A_2454_MXZ01.StFault := FALSE;
   A_2454_MXZ01.StStartedRev := FALSE;
   A_2454_MXZ01.InOutManSlow := FALSE;
   A_2454_MXZ01.InOutManRev := FALSE;
   A_2454_MXZ01.OutAlarmNrLog := 0;
   A_2454_MXZ01.Par.ParObjectNo := 1711;
   A_2454_MXZ01.Par.ParMsgType := 7053;
   A_2454_MXZ01.Par.ParHornCode := 0;
   A_2454_MXZ01.Par.ParLogOff := FALSE;
   A_2454_MXZ01.Par.ParManual := TRUE;
   A_2454_MXZ01.Par.ParRestartDelay := FALSE;
   A_2454_MXZ01.Par.Par2Speed := FALSE;
   A_2454_MXZ01.Par.ParHeavyStartup := FALSE;
   A_2454_MXZ01.Par.spare45 := FALSE;
   A_2454_MXZ01.Par.spare46 := FALSE;
   A_2454_MXZ01.Par.OutEdgeFaultReset := FALSE;
   A_2454_MXZ01.Par.OutDelayFault := FALSE;
   A_2454_MXZ01.Par.OutFlagFaultDev := FALSE;
   A_2454_MXZ01.Par.ParMonTime := 20;
   A_2454_MXZ01.Par.ParStartingTime := 20;
   A_2454_MXZ01.Par.ParStoppingTime := 0;
   A_2454_MXZ01.Par.ParIdlingTime := 0;
   A_2454_MXZ01.Par.ParDelayTime := 10;
   A_2454_MXZ01.Par.OutMonTime := 0;
   A_2454_MXZ01.Par.OutTransitionTime := 0;
   A_2454_MXZ01.Par.OutDelayTime := 0;
   A_2454_MXZ01.Par.InOutManPulseLen := 0;
   A_2455_MXZ01.StCode := 0;
   A_2455_MXZ01.InEnableRev := FALSE;
   A_2455_MXZ01.InEnableFwd := FALSE;
   A_2455_MXZ01.InSlow := FALSE;
   A_2455_MXZ01.InpRunSlow := FALSE;
   A_2455_MXZ01.InpRunFast := FALSE;
   A_2455_MXZ01.InpRunRev := FALSE;
   A_2455_MXZ01.InpRunFwd := FALSE;
   A_2455_MXZ01.InpFaultDev := FALSE;
   A_2455_MXZ01.CmdOff := FALSE;
   A_2455_MXZ01.CmdOn := FALSE;
   A_2455_MXZ01.CmdNext := FALSE;
   A_2455_MXZ01.CmdFaultReset := FALSE;
   A_2455_MXZ01.InLocal := FALSE;
   A_2455_MXZ01.InManual := FALSE;
   A_2455_MXZ01.InReport := FALSE;
   A_2455_MXZ01.InSeqStop := FALSE;
   A_2455_MXZ01.InHWStop := FALSE;
   A_2455_MXZ01.InDPFault := FALSE;
   A_2455_MXZ01.OutIdling := FALSE;
   A_2455_MXZ01.OutpRunSlow := FALSE;
   A_2455_MXZ01.OutpRunFast := FALSE;
   A_2455_MXZ01.OutpRunRev := FALSE;
   A_2455_MXZ01.OutpRunFwd := FALSE;
   A_2455_MXZ01.OutpFaultReset := FALSE;
   A_2455_MXZ01.StStopped := FALSE;
   A_2455_MXZ01.StStarting := FALSE;
   A_2455_MXZ01.StStartedFwd := FALSE;
   A_2455_MXZ01.StStopping := FALSE;
   A_2455_MXZ01.StFault := FALSE;
   A_2455_MXZ01.StStartedRev := FALSE;
   A_2455_MXZ01.InOutManSlow := FALSE;
   A_2455_MXZ01.InOutManRev := FALSE;
   A_2455_MXZ01.OutAlarmNrLog := 0;
   A_2455_MXZ01.Par.ParObjectNo := 17712;
   A_2455_MXZ01.Par.ParMsgType := 7053;
   A_2455_MXZ01.Par.ParHornCode := 0;
   A_2455_MXZ01.Par.ParLogOff := FALSE;
   A_2455_MXZ01.Par.ParManual := TRUE;
   A_2455_MXZ01.Par.ParRestartDelay := FALSE;
   A_2455_MXZ01.Par.Par2Speed := FALSE;
   A_2455_MXZ01.Par.ParHeavyStartup := FALSE;
   A_2455_MXZ01.Par.spare45 := FALSE;
   A_2455_MXZ01.Par.spare46 := FALSE;
   A_2455_MXZ01.Par.OutEdgeFaultReset := FALSE;
   A_2455_MXZ01.Par.OutDelayFault := FALSE;
   A_2455_MXZ01.Par.OutFlagFaultDev := FALSE;
   A_2455_MXZ01.Par.ParMonTime := 20;
   A_2455_MXZ01.Par.ParStartingTime := 20;
   A_2455_MXZ01.Par.ParStoppingTime := 0;
   A_2455_MXZ01.Par.ParIdlingTime := 0;
   A_2455_MXZ01.Par.ParDelayTime := 10;
   A_2455_MXZ01.Par.OutMonTime := 0;
   A_2455_MXZ01.Par.OutTransitionTime := 0;
   A_2455_MXZ01.Par.OutDelayTime := 0;
   A_2455_MXZ01.Par.InOutManPulseLen := 0;
END_DATA_BLOCK

